FUNCTION_BLOCK FB_Observable_UDINT EXTENDS FB_AbstractObservable
VAR
    _nVal:              UDINT;
END_VAR

METHOD FB_init : BOOL
VAR_INPUT
    bInitRetains:       BOOL; // if TRUE, the retain variables are initialized (warm start / cold start)
    bInCopyCode:        BOOL;  // if TRUE, the instance afterwards gets moved into the copy code (online change)
    bAutoNotify:        BOOL;
END_VAR
THIS^._nTypeClass := __SYSTEM.TYPE_CLASS.TYPE_UDINT;
END_METHOD

METHOD  Notify : I_Observable
VAR
    i:      UDINT;
END_VAR
Notify := THIS^;

IF THIS^.nObserverCount <= 0 THEN
    RETURN;
END_IF

FOR i := 0 TO THIS^.nLastIdx DO
    THIS^.pipObserver[i].Update(THIS^._nVal);
END_FOR
END_METHOD

METHOD  NotifyLast : I_Observable
NotifyLast := THIS^;

IF THIS^.nObserverCount <= 0 THEN
    RETURN;
END_IF

THIS^.pipObserver[THIS^.nLastIdx].Update(THIS^._nVal);
END_METHOD

PROPERTY nValue32 : UDINT
GET
nValue32 := THIS^._nVal;
END_GET
SET
THIS^._nVal := nValue32;

IF THIS^._bAutoNotify THEN
    THIS^.Notify();
END_IF
END_SET
END_PROPERTY

END_FUNCTION_BLOCK

(* stored: Version 1.1.0.1, ProductVersion 3.1.4024.12
   POU FB_Observable_UDINT: Id {d0660e49-c775-410d-a0a1-9e032074c447}, SpecialFunc None
   Method FB_init: Id {1e068f87-8594-0c5a-1471-1ede03cfb060}
   Method Notify: Id {7bf07f9f-9a73-4cb8-8e42-b2f4644a79b1}
   Method NotifyLast: Id {146a901e-f8dc-4d96-b1cb-110d36bf9c72}
   Property nValue32: Id {1b1add70-3051-4ef1-935b-e2d6c1d98d7e}
   Get Get: Id {632ceaa0-021f-4af2-aa9d-7e6a21040b3d}
   Set Set: Id {79fae39c-6271-4ab4-972b-e43b59cbba29} *)
